{attribute 'qualified_only'}
{attribute 'strict'}
TYPE E_Xelectrix_GridState :
(
	eNoDataReceived := 0,
	eOff := 1,
	eIslandMode := 2,
	eOnline := 3,
	eError := 4
);
END_TYPE

(* stored: Version 1.1.0.1, ProductVersion 3.1.4024.6
   DUT E_Xelectrix_GridState: Id {3c818955-eefb-42f6-a113-d9df22a3641d} *)
